TYPE
    ST_HMI_MachineStatus :
    STRUCT
        Axes      : ST_AXES_STATUS;	  //馬達狀態
        Cylinders : ST_CylinderStatus;//汽缸狀態
        Motor     : ST_MotorStatus;	  //軌道狀態
    END_STRUCT
END_TYPE

(* stored: Version 1.1.0.1, ProductVersion 3.1.4024.13
   DUT ST_HMI_MachineStatus: Id {40bc4766-38d4-4a8c-8f9f-836706fd45b7} *)
